PROGRAM Read_ID
VAR
	PrimeMover_ID			: STRING := '2';
	Trailer_ID_Lead AT %I*	: UINT;
	Trailer_ID_Rear AT %I*	: UINT;
END_VAR

;

END_PROGRAM

(* stored: Version 1.1.0.1, ProductVersion 3.1.4024.6
   POU Read_ID: Id {e1372c7c-abe8-4077-94d5-6aa297d659bb}, SpecialFunc None *)
